{attribute addProperty BoxType "EK1100-0000-0018"}
{attribute addProperty Id "Beckhoff_EP7xxxEK1122Beckhoff_EP7xxxEK1122_CDE5BCF8150051875.625"}
{attribute addProperty CRC "2453673006"}
{attribute addProperty SizeInBites "15005"}
{attribute addProperty SizeInBytes "1875.625"}
TYPE Beckhoff_EP7xxx_9240142E EXTENDS EK1100_179A0949 :
STRUCT
	{attribute addProperty Name "Beckhoff_EP7xxxEK1122"}
	Beckhoff_EP7xxxEK1122 : Beckhoff_EP7xxxEK1122_CDE5BCF8;
END_STRUCT
END_TYPE

(* stored: Version 1.2.0.0, ProductVersion 3.1.4024.9
   DUT Beckhoff_EP7xxx_9240142E: Id {a2d114a9-11ad-4d38-b15d-e18dc91ebe7d} *)
